TYPE HMIMovementForkInterface :
STRUCT
	ForkMovementSettingLines	:	ARRAY [1..3] of HMISettingLineInterface;
END_STRUCT
END_TYPE

(* stored: Version 1.1.0.1
   DUT HMIMovementForkInterface: Id {78f23466-a8b8-4bc5-9f92-db87a0e2d99a} *)
